FUNCTION_BLOCK Plant
  (* Standard: 61499-2 *)
  (* Version 0.1, 2017-00-23, hpea485, UOA *)
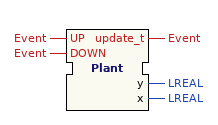
  EVENT_INPUT
    UP;
    DOWN;
  END_EVENT
  EVENT_OUTPUT
    update_t;
  END_EVENT
  VAR_OUTPUT
    y : LREAL;
    x : LREAL;
  END_VAR
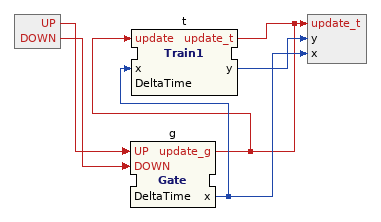
  FBS
    g : Gate;
    t : Train1;
  END_FBS
  EVENT_CONNECTIONS
    UP TO g.UP;
    DOWN TO g.DOWN;
    t.update_t TO update_t;
    g.update_g TO update_t;
    g.update_g TO t.update;
  END_CONNECTIONS
  DATA_CONNECTIONS
    t.y TO y;
    g.x TO x;
    g.x TO t.x;
  END_CONNECTIONS
END_FUNCTION_BLOCK
